(* CoDeSys 2.3.9.41 project: lab6.pro *)
(* Libraries: STANDARD.LIB 5.6.98 11:03:02 *)

(* Task configuration *)
TASK Standard (PRIORITY := 0, INTERVAL := T#1ms);
	MAIN
END_TASK

(* Global variable list: Global_Variables *)
VAR_GLOBAL
	PERIOD : REAL := 0.001;
END_VAR

(* Data type *)
TYPE PID_Parameter_Struct :
STRUCT
	Kp : REAL;
	Ti: REAL;
	Td : REAL;
	N : UINT;
	ARW : BOOL;
	Umin : REAL;
	Umax : REAL;
END_STRUCT
END_TYPE

(* Data type *)
TYPE PT1T2_Parameter_Strukt :
STRUCT
	K : REAL;
	T1 : REAL;
	T2: REAL;
END_STRUCT
END_TYPE

(* Data type *)
TYPE System_Modus_Enum:
(
	System_Init,
	System_Run
);
END_TYPE

(* POU MAIN, ST *)
PROGRAM MAIN
VAR
	paramS : PT1T2_Parameter_Strukt;
	paramPid : PID_Parameter_Struct;
	Modus : System_Modus_Enum := System_Init;
	PID_1 : PID;
	S_1 : Strecke;
	Ref : REAL := 0;
	u : REAL;
	y : REAL;
	e : REAL;
END_VAR
CASE Modus OF
System_Init:
	paramS.K := 10;
	paramS.T1 := 0.1;
	paramS.T2 := 0.01;
	paramPid.Kp := 1/paramS.K;
	paramPid.Ti := paramS.T1;
	paramPid.Td := paramS.T2;
	paramPid.N := 10;
	PID_1(input_e := 0, input_y := 0, param := paramPid, modus := Modus);
	S_1(input := 0, param := paramS, modus := Modus);
	Modus := System_Run;

System_Run:
	e := Ref - y;
	PID_1(input_e := e, input_y := y, param := paramPid, modus := Modus);
	u := PID_1.out;
	S_1(input := u, param := paramS, modus := Modus);
	y := S_1.out;
END_CASE
END_PROGRAM

(* POU PID, ST *)
FUNCTION_BLOCK PID
VAR_INPUT
	input_e : REAL;
	input_y : REAL;
	param : PID_Parameter_Struct;
	modus : System_Modus_Enum;
END_VAR

VAR_OUTPUT
	out: REAL;
END_VAR

VAR
	p : REAL;
	i : REAL;
	d : REAL;
	Ki : REAL;
	Kd : REAL;
	input_e_z1 : REAL;
	input_y_z1 : REAL;
	i_z1 : REAL;
	d_z1 : REAL;
	out_z1 : REAL;
	out_z2 : REAL;
END_VAR
CASE modus OF
System_init:
	Ki := param.Kp * PERIOD / (2 * param.Ti);
	Kd := 1/(1/param.N + PERIOD/(2 * param.Td));
	Kd := param.N * PERIOD + param.Td;
	Kd := 1 / (1 + (param.N * PERIOD) / (param.Td));

System_run:
	p := input_e * param.Kp;
	i   := i_z1 +   Ki * (input_e + input_e_z1);
	d := (-input_y * param.N * param.Td + input_y_z1 * param.Td + out_z1 * param.Td) / (Kd);
	d := Kd * (d_z1 + (input_y - input_y_z1) * param.N);

	out := p + i + d;

	input_e_z1 := input_e;
	input_y_z1 := input_y;
	i_z1 := i;
	d_z1 := d;
	out_z2 := out_z1;
	out_z1 := out;
END_CASE
END_FUNCTION_BLOCK

(* POU Strecke, ST *)
FUNCTION_BLOCK Strecke
VAR_INPUT
	input : REAL;
	param : PT1T2_Parameter_Strukt;
	modus : System_Modus_Enum;
END_VAR

VAR_OUTPUT
	out : REAL;
END_VAR

VAR
	b0 : REAL;
	b1 : REAL;
	c1 : REAL;
	c2 : REAL;
	a1 : REAL;
	a2 : REAL;
	lastY : REAL;
	lastLastY: REAL;
	lastU : REAL;
	lastLastU: REAL;
END_VAR
CASE modus OF
System_Init:
	a1 := EXP(-PERIOD/param.T1);
	a2 := EXP(-PERIOD/param.T2);
	b0 :=(param.K/(param.T1-param.T2)) * (param.T1*(1- a1)-param.T2*(1- a2));
	b1 :=(param.K/(param.T1-param.T2)) * (param.T2*a1*(1- a2)-param.T1*a2*(1- a1));
	c1 := -(a1+a2);
	c2 := a1 * a2;

System_Run:
	out := b0 * lastU + b1*lastLastU - c1 * LastY - c2 * LastLastY;
	lastLastU := lastU;
	lastU := input;

	lastLastY := lastY;
	lastY := out;
END_CASE
END_FUNCTION_BLOCK
